FUNCTION_BLOCK fb_zoh_real

VAR_INPUT
	x		:REAL;
END_VAR

VAR_OUTPUT
	y		:REAL;
	last	:REAL;	
END_VAR

VAR

END_VAR


y:=last;
last:=x;

END_FUNCTION_BLOCK

(* stored: Version 1.1.0.1, ProductVersion 3.1.0.26
   POU fb_zoh_real: Id {4dfcd6b8-2520-44fd-8b5a-43fdd1c76784} *)
